{attribute addProperty BoxType "EK1100-0000-0018"}
{attribute addProperty Id "Beckhoff_ELM3xxx_0030EK1122Beckhoff_ELM3xxx_0030EK1122_7F195F23162A_0001_ELM3002_0030_0017ELM3002_08F8D9E433842.25A_0002_ELM3002_0030_0018ELM3002_08F8D9E433842.25A_0003_ELM3004_0030_0018ELM3004_B740F21646658.25A_0004_ELM3004_0030_0019ELM3004_B740F21646658.25A_0005_ELM3502_0030_0019ELM3502_08F8D9E433842.25A_0006_ELM3504_0030_0019ELM3504_B740F21646658.25"}
{attribute addProperty CRC "2263615264"}
{attribute addProperty SizeInBites "2428"}
{attribute addProperty SizeInBytes "303.5"}
TYPE Beckhoff_ELM3xxx_0030_86EC0720 EXTENDS EK1100_179A0949 :
STRUCT
	{attribute addProperty Name "Beckhoff_ELM3xxx_0030EK1122"}
	Beckhoff_ELM3xxx_0030EK1122 : Beckhoff_ELM3xxx_0030EK1122_7F195F23;
	{attribute addProperty Name "A_0001_ELM3002_0030_0017"}
	A_0001_ELM3002_0030_0017 : ELM3002_08F8D9E4;
	{attribute addProperty Name "A_0002_ELM3002_0030_0018"}
	A_0002_ELM3002_0030_0018 : ELM3002_08F8D9E4;
	{attribute addProperty Name "A_0003_ELM3004_0030_0018"}
	A_0003_ELM3004_0030_0018 : ELM3004_B740F216;
	{attribute addProperty Name "A_0004_ELM3004_0030_0019"}
	A_0004_ELM3004_0030_0019 : ELM3004_B740F216;
	{attribute addProperty Name "A_0005_ELM3502_0030_0019"}
	A_0005_ELM3502_0030_0019 : ELM3502_08F8D9E4;
	{attribute addProperty Name "A_0006_ELM3504_0030_0019"}
	A_0006_ELM3504_0030_0019 : ELM3504_B740F216;
END_STRUCT
END_TYPE

(* stored: Version 1.2.0.0, ProductVersion 3.1.4024.9
   DUT Beckhoff_ELM3xxx_0030_86EC0720: Id {a80d2239-5c4a-424d-b3c9-1c81de950b9d} *)
